TYPE LIMIT_STATES :
(
	NO_LENSES := 0,
	XRT_ONLY  := 1,
	MFX_ONLY  := 2,
	PREFOCUS := 3
	
);
END_TYPE

(* stored: Version 1.1.0.1, ProductVersion 3.1.4018.5
   DUT LIMIT_STATES: Id {592e01d0-0d36-41c4-a333-b1d9bba78f5b} *)
